FUNCTION_BLOCK Controller (* Basic Function Block Type *)
  (* Standard: 61499-2 *)
  (* Version 0.3, 2009-09-15, JHC, Holobloc Inc, Changed transition priorities. *)
  (* Version 0.2, 2003-12-04, JHC, Rockwell Automation, Renamed for better indexing. *)
  (* Version 0.1, 2002-11-05, JHC, Rockwell Automation, Corrected missing ST element in Algorithm REQ. *)
  (* Version 0.0, 2000-05-30, JHC, Rockwell Automation *)
  (* Compiler header: package fb.rt.template; *)
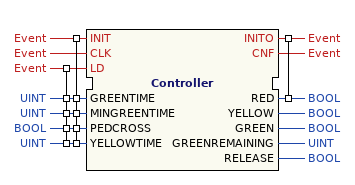
  EVENT_INPUT
    INIT WITH GREENTIME, MINGREENTIME, PEDCROSS, YELLOWTIME; (* Initialization Request *)
    CLK; (* Normal Execution Request *)
    LD WITH GREENTIME, MINGREENTIME, PEDCROSS, YELLOWTIME;
  END_EVENT
  EVENT_OUTPUT
    INITO WITH RED; (* Initialization Confirm *)
    CNF;
  END_EVENT
  VAR_INPUT
    GREENTIME : UINT;
    MINGREENTIME : UINT;
    PEDCROSS : BOOL;
    YELLOWTIME : UINT;
  END_VAR
  VAR_OUTPUT
    RED : BOOL; (* Output event qualifier *)
    YELLOW : BOOL;
    GREEN : BOOL;
    GREENREMAINING : UINT;
    RELEASE : BOOL;
  END_VAR
  VAR
    MINGREENTIMEIN : UINT;
    YELLOWTIMEIN : UINT;
    GREENTIMEIN : UINT;
  END_VAR
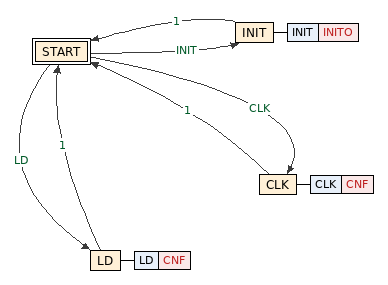
  EC_STATES
    START; (* Initial State *)
    INIT : INIT -> INITO; (* Initialization *)
    CLK : CLK -> CNF; (* Normal execution *)
    LD : LD -> CNF;
  END_STATES
  EC_TRANSITIONS
    INIT TO START := 1;
    START TO CLK := CLK;
    START TO INIT := INIT;
    CLK TO START := 1;
    START TO LD := LD;
    LD TO START := 1;
  END_TRANSITIONS
  ALGORITHM INIT IN ST: (* Initialization algorithm *)
RED:=FALSE;
YELLOW:=FALSE;
GREEN:=FALSE;
MINGREENTIMEIN:=100;
YELLOWTIMEIN:=100;
GREENTIMEIN:=100;
RELEASE:=FALSE;
  END_ALGORITHM
  ALGORITHM CLK IN ST: (* Normally executed algorithm *)
IF PEDCROSS THEN
	IF MINGREENTIMEIN<=0 THEN
  		GREEN:=FALSE;
  		YELLOW:=TRUE;
  		RED:=FALSE;
  		GREENTIMEIN:=0;
	END_IF;
END_IF;
IF GREENTIMEIN>0 THEN
	GREENTIMEIN := GREENTIMEIN - 1;
    MINGREENTIMEIN:= MINGREENTIMEIN - 1;
    GREEN:=TRUE;
	YELLOW:= FALSE;
    RED:=FALSE;
END_IF;
GREENREMAINING:=GREENTIMEIN;
IF GREENTIMEIN=0 THEN
    GREEN:=FALSE;
	YELLOW:= TRUE;
    RED:=FALSE;
	IF YELLOWTIMEIN>0 THEN
		YELLOWTIMEIN:= YELLOWTIMEIN - 1;
	END_IF;
 IF YELLOWTIMEIN=0 THEN
      GREEN:=FALSE;
      YELLOW:=FALSE;
	  RED:=TRUE;
	  RELEASE:=TRUE;
	END_IF;
END_IF;
  END_ALGORITHM
  ALGORITHM LD IN ST:
GREEN:=TRUE;
YELLOW:=FALSE;
RED:=FALSE;
MINGREENTIMEIN:=MINGREENTIME;
YELLOWTIMEIN:=YELLOWTIME;
GREENTIMEIN:=GREENTIME;
GREENREMAINING:=GREENTIME;
RELEASE:=FALSE;
  END_ALGORITHM
END_FUNCTION_BLOCK
